% RSLogix 500 project Filmore Piru HPW 2015.RSS, saved by version 11.00.00.00 %
PROJECT "UNTITLED"    % processor: MicroLogix 1000 %

PROGRAM FILES
  LAD 2 "MAIN_PROG"  14 rungs
  LAD 3 "USER_FAULT"  1 rungs
  LAD 4 "HSC_INT"  1 rungs
  LAD 5 "STI_INT"  1 rungs
  LAD 6, 7, 8, 9, 10, 11, 12, 13, 14, 15, 16: only END

DATA FILES
  O0 OUTPUT  1 elements
  I1 INPUT  2 elements
  S2 STATUS  33 elements
  B3 BINARY  32 elements
  T4 TIMER  40 elements
  C5 COUNTER  32 elements
  R6 CONTROL  16 elements
  N7 INTEGER  105 elements

LADDER 2 "MAIN_PROG"
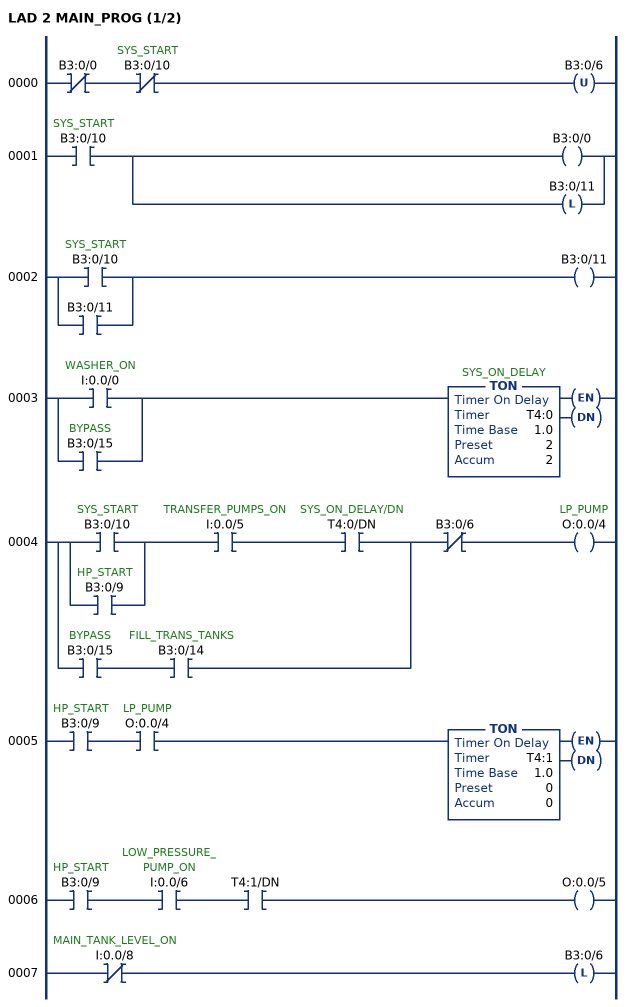
% Rung: 0 %
SOR XIO B3:0/0 XIO B3:0/10 OTU B3:0/6 EOR
%   B3:0/10  SYS_START %
% Rung: 1 %
SOR XIC B3:0/10 BST OTE B3:0/0 NXB OTL B3:0/11 BND EOR
%   B3:0/10  SYS_START %
% Rung: 2 %
SOR BST XIC B3:0/10 NXB XIC B3:0/11 BND OTE B3:0/11 EOR
%   B3:0/10  SYS_START %
% Rung: 3 %
SOR BST XIC I:0.0/0 NXB XIC B3:0/15 BND TON T4:0 1.0 2 2 EOR
%   I:0.0/0  WASHER_ON %
%   B3:0/15  BYPASS %
%   T4:0  SYS_ON_DELAY %
% Rung: 4 %
SOR BST BST XIC B3:0/10 NXB XIC B3:0/9 BND XIC I:0.0/5 XIC T4:0/DN NXB XIC B3:0/15 XIC B3:0/14 BND XIO B3:0/6 OTE O:0.0/4 EOR
%   B3:0/10  SYS_START %
%   B3:0/9  HP_START %
%   I:0.0/5  TRANSFER_PUMPS_ON %
%   T4:0  SYS_ON_DELAY %
%   B3:0/15  BYPASS %
%   B3:0/14  FILL_TRANS_TANKS %
%   O:0.0/4  LP_PUMP %
% Rung: 5 %
SOR XIC B3:0/9 XIC O:0.0/4 TON T4:1 1.0 0 0 EOR
%   B3:0/9  HP_START %
%   O:0.0/4  LP_PUMP %
% Rung: 6 %
SOR XIC B3:0/9 XIC I:0.0/6 XIC T4:1/DN OTE O:0.0/5 EOR
%   B3:0/9  HP_START %
%   I:0.0/6  LOW_PRESSURE_PUMP_ON %
% Rung: 7 %
SOR XIO I:0.0/8 OTL B3:0/6 EOR
%   I:0.0/8  MAIN_TANK_LEVEL_ON %

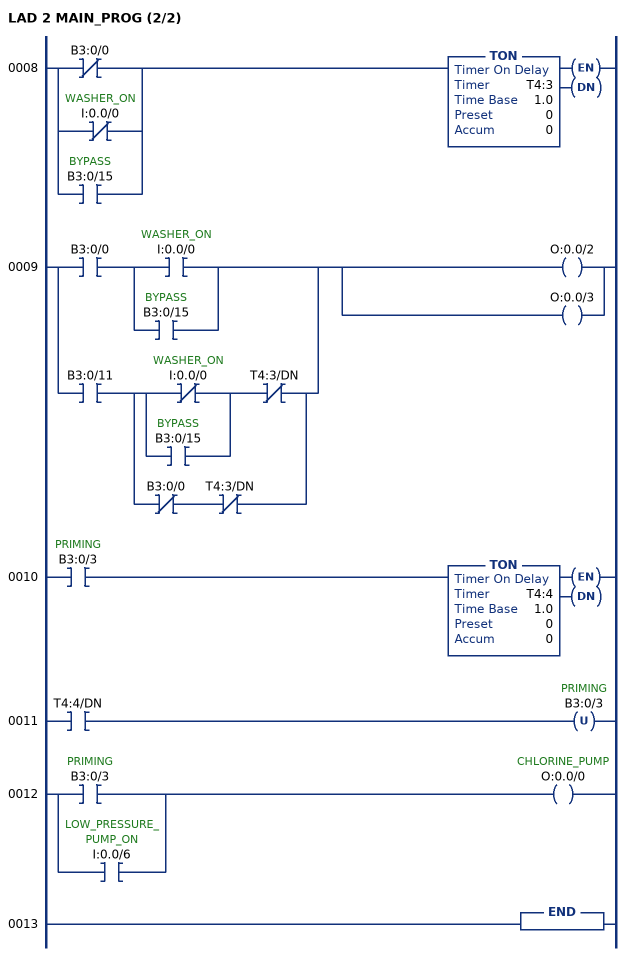
% Rung: 8 %
SOR BST XIO B3:0/0 NXB BST XIO I:0.0/0 NXB XIC B3:0/15 BND BND TON T4:3 1.0 0 0 EOR
%   I:0.0/0  WASHER_ON %
%   B3:0/15  BYPASS %
% Rung: 9 %
SOR BST XIC B3:0/0 BST XIC I:0.0/0 NXB XIC B3:0/15 BND NXB XIC B3:0/11 BST BST XIO I:0.0/0 NXB XIC B3:0/15 BND XIO T4:3/DN NXB XIO B3:0/0 XIO T4:3/DN BND BND BST OTE O:0.0/2 NXB OTE O:0.0/3 BND EOR
%   I:0.0/0  WASHER_ON %
%   B3:0/15  BYPASS %
% Rung: 10 %
SOR XIC B3:0/3 TON T4:4 1.0 0 0 EOR
%   B3:0/3  PRIMING %
% Rung: 11 %
SOR XIC T4:4/DN OTU B3:0/3 EOR
%   B3:0/3  PRIMING %
% Rung: 12 %
SOR BST XIC B3:0/3 NXB XIC I:0.0/6 BND OTE O:0.0/0 EOR
%   B3:0/3  PRIMING %
%   I:0.0/6  LOW_PRESSURE_PUMP_ON %
%   O:0.0/0  CHLORINE_PUMP %
% Rung: 13 %
SOR END EOR

OTHER DOCUMENTED ADDRESSES
  B3:0/2  NO_PRIMING
  I:0.0/7  HIGH_PRESS_PUMP_ON
  I:0.0/9  TRANSFER_TANK_LEVEL
  T4:0.PRE  START_DELAY
  T4:1.PRE  HP_START_DELAY
  T4:3.PRE  TRANS_OFF_DELAY
  T4:4.PRE  PRIME_DURATION
  T4:6/EN  CHL_PUMPS_ON

DATA TABLE (non-zero values as saved)
DATA B3
% B3:0 % 0X0C01 0X0000 0X0000 0X0000 0X0000 0X0000 0X0000 0X0000 0X0000 0X0000
DATA T4
% .PRE .ACC %
% T4:0 % 2 2
% T4:2 % 2 0
% T4:5 % 10 0
% T4:6 % 50 0
